Universal Robots PolyScope program: modbus.urp

Program modbus (installation=default directory=/home/ur/ursim-current/programs createdIn=5.12.6.1102099 lastSavedIn=5.12.6.1102099 robotSerialNumber=20195299999)
Calibrated DH parameters: a=[0, -0.6127, -0.57155, 0, 0, 0]; d=[0.1807, 0, 0, 0.17415, 0.11985, 0.11655]; alpha=[1.570796, 0, 0, 1.570796, -1.570796, 0]; deltaTheta=[0, 0, 0, 0, 0, 0]
Robot Program (runOnlyOnce=false)
  var_2 := MODBUS_1
  Wait Sleep waitTime=2
  var_1 := MODBUS_2
  Wait Sleep waitTime=2
